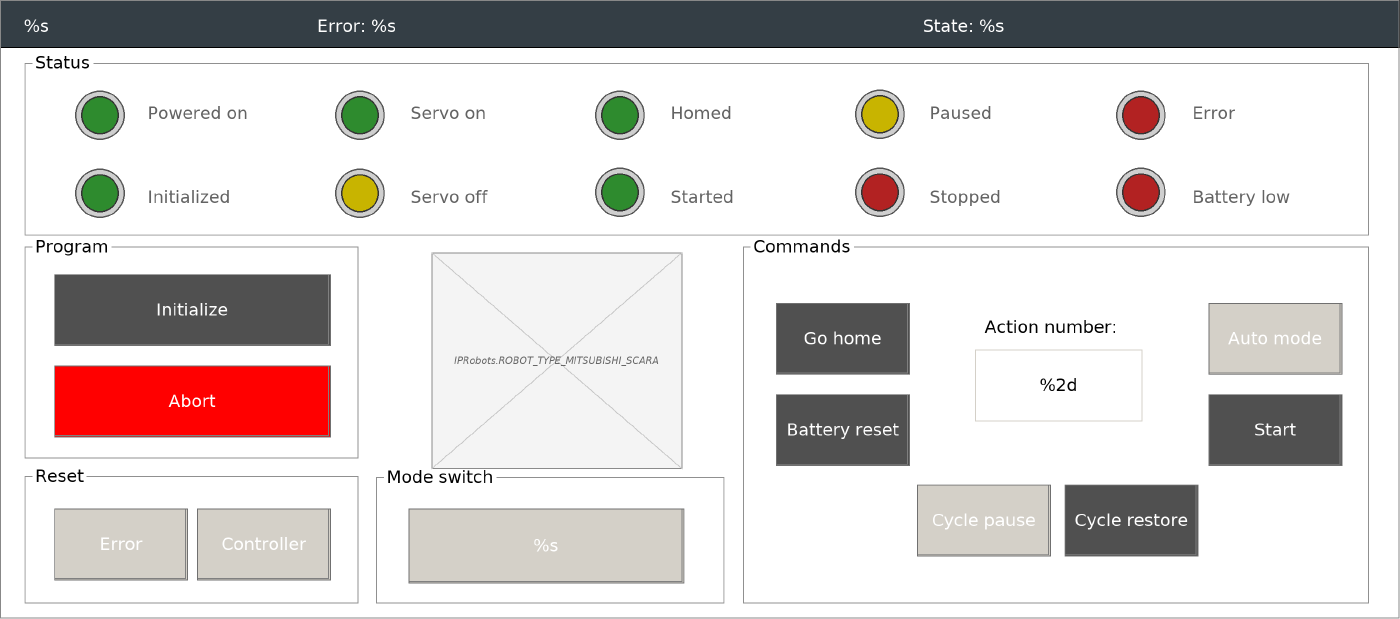
VISUALIZATION SingleRobot  // 1470x650
VAR_IN_OUT
	stRobot		: ST_VisuCtrlRobotFrame;
END_VAR
    Rectangle (0,0 1470x50)
    Textfield (22,10 296x35), "%s", text variable: stRobot.sName
    Textfield (966,10 498x35), "State: %s", text list: 'TL_SingleRobotState', text index: stRobot.eRobotState
    Textfield (330,10 628x35), "Error: %s", text variable: stRobot.sErrorDescription
    Image (453,265 263x227), image: IPRobots.ROBOT_TYPE_MITSUBISHI_SCARA
        p84334746: stRobot.sRobotImage
    GroupBox (26,58 1411x189), "Status"
        Lamp1 (595,33 60x60), variable: stRobot.bIsHomed, style: Lamp-Lamp1-Green
        Lamp1 (595,114 60x60), variable: stRobot.bStarted, style: Lamp-Lamp1-Green
        Rectangle (675,37 150x48), "Homed"
        Rectangle (675,125 150x48), "Started"
        Lamp1 (1142,114 60x60), variable: stRobot.bBatteryLow, style: Lamp-Lamp1-Red
        Rectangle (1223,125 150x48), "Battery low"
        Lamp1 (1142,33 60x60), variable: stRobot.bError, style: Lamp-Lamp1-Red
        Rectangle (1223,37 150x48), "Error"
        Lamp1 (49,33 60x60), variable: stRobot.bPowerOn, style: Lamp-Lamp1-Green
        Lamp1 (49,115 60x60), variable: stRobot.bInit, style: Lamp-Lamp1-Green
        Rectangle (126,37 150x48), "Powered on"
        Rectangle (126,125 150x48), "Initialized"
        Rectangle (402,37 150x48), "Servo on"
        Rectangle (402,125 150x48), "Servo off"
        Lamp1 (322,33 60x60), variable: stRobot.bServoOn, style: Lamp-Lamp1-Green
        Lamp1 (322,115 60x60), variable: stRobot.bServoOff, style: Lamp-Lamp1-Yellow
        Rectangle (947,37 150x48), "Paused"
        Rectangle (947,125 150x48), "Stopped"
        Lamp1 (868,32 60x60), variable: stRobot.bPaused, style: Lamp-Lamp1-Yellow
        Lamp1 (868,114 60x60), variable: stRobot.bStopped, style: Lamp-Lamp1-Red
    GroupBox (26,251 350x230), "Program"
        Button (31,37 290x75), "Initialize", input disabled if: stRobot.bInitButtonDisable
            tap stRobot.btnInit
        Button (31,133 290x75), "Abort", input disabled if: stRobot.bUninitialized
            tap stRobot.btnAbort
    GroupBox (26,492 350x141), "Reset"
        Button (31,42 140x75), "Error"
            tap stRobot.btnErrorReset
        Button (181,42 140x75), "Controller"
            tap stRobot.btnControllerReset
    GroupBox (780,251 657x382), "Commands"
        Button (489,163 140x75), "Start", input disabled if: stRobot.bActionButtonDisable
            tap stRobot.btnDoAction
        Button (35,67 140x75), "Go home", input disabled if: stRobot.bHomeButtonDisable
            tap stRobot.btnGoHome
        Button (489,67 140x75), "Auto mode", input disabled if: stRobot.bAutoButtonDisable
            tap stRobot.btnGoAuto
        Button (35,163 140x75), "Battery reset", input disabled if: stRobot.bAutoButtonDisable
        Rectangle (251,80 160x25), "Action number:"
        Button (338,258 140x75), "Cycle restore", input disabled if: stRobot.bRestoreCycleButtonDisable
            tap stRobot.btnRestoreCycle
        Button (183,258 140x75), "Cycle pause", input disabled if: stRobot.bPausingButtonDisable
            tap stRobot.btnCyclePause
        Textfield (244,116 175x75), "%2d", text variable: stRobot.iActionNumber, input disabled if: stRobot.bActionButtonDisable
            OnMouseClick: write the text variable via VisuDialogs.Numpad, min 13, max 100
    GroupBox (395,493 365x140), "Mode switch", invisible if: stRobot.bModeSwitchButtonDisabled
        Button (34,41 289x78), "%s", input disabled if: stRobot.bInit, text list: 'TL_ModeSwitchState', text index: stRobot.bModeSwitchState
            toggle stRobot.btnModeSwitch
END_VISUALIZATION

(* stored: Version 1.1.0.1, ProductVersion 3.1.4024.12
   Visu SingleRobot: Id {b8e04ad4-db2f-48de-bc32-f9a7581dff05} *)
